// TIA Portal V16 export
// export: Created 2022-07-21T09:35:35.040371Z, ExportSetting WithDefaults, DisplayName Totally Integrated Automation Portal, DisplayVersion V16 Update 4, DisplayName TIA Portal Version Control Interface, DisplayVersion V16 Update 2, DisplayName TIA Portal Openness, DisplayVersion V16 Update 4, DisplayName SINAMICS Startdrive Advanced, DisplayVersion V16 Update 5, DisplayName SINAMICS Startdrive G130, G150, S120, S150, SINAMICS MV, S210, DisplayVersion V16 Update 5, DisplayName SINAMICS Startdrive G110M, G120, G120C, G120D, G120P, G115D, DisplayVersion V16 Update 5, DisplayName STEP 7 Professional, DisplayVersion V16 Update 4, DisplayName STEP 7 Safety, DisplayVersion V16, DisplayName WinCC Advanced, DisplayVersion V16 Update 4
FUNCTION_BLOCK "fbValve"   // FB702, LAD
TITLE = Valve / Obsługa zaworu
{ S7_Optimized_Access := 'TRUE' }
AUTHOR : a32thzz
VERSION : 0.1
// In this block alarms, statuses and commands for electrovalves are generated / Ten blok służy do generowania alarmów, statusów i wysyłania komend dla siłowników kontrolowanych przez elektrozawory.
// stored: AutoNumber false, IsIECCheckEnabled false, IsRetainMemResEnabled false, MemoryReserve 100, SetENOAutomatically false, UDAEnableTagReadback false
   VAR_INPUT
      inPeripheryOK : Bool;   // Zezwolenie od peryferiów (PN, Elektryka)
      inHomeLS : Bool;   // Czujnik pozycji bazowej / Home position sensor
      inWorkLS : Bool;   // Czujnik pozycji roboczej / Work position sensor
      inAutoHome : Bool;   // Krok sekwencji "do pozycji bazowej" / Move to home position
      inAutoWork : Bool;   // Krok sekwencji "do pozycji roboczej" / Move to work position
      inHold : Bool := true;   // Podtrzymanie zasilania elektrozaworu podczas ruchu do pozycji / Hold electrovalve power supply during movement
      inJog : Bool := true;   // Podtrzymanie zasilania elektrozaworu po osiągnięciu pozycji końcowej / Hold electrovalve power supply after reaching position
      inDelayPTAlm0 : Time := T#1s;   // Czas opóźnienia dla alarmu 0 / alarm delay 0
      inDelayPTAlm1 : Time := T#1s;   // Czas opóźnienia dla alarmu 1 / alarm delay 1
      inDelayPTAlm2 : Time := T#1s;   // Czas opóźnienia dla alarmu 2 / alarm delay 2
      inDelayPTAlm3 : Time := T#1s;   // Czas opóźnienia dla alarmu 3 / alarm delay 3
      inDelayPTAlm4 : Time := T#1s;   // Czas opóźnienia dla alarmu 4 / alarm delay 4
      inDelayPTAlm5 : Time := T#1s;   // Czas opóźnienia dla alarmu 5 / alarm delay 5
      inAlmMask : Word := W#16#FFE0;   // Maskowanie alarmów
      inGroup : "typeGroup";   // Grupa do której przypisany jest zawór / Valve group
   END_VAR
   VAR_OUTPUT
      ouHomeSV : Bool;   // Elektrozawór dla pozycji bazowej / Electrovalve to home porisiton
      ouWorkSV : Bool;   // Elektrozawór dla pozycji roboczej / Electrovalve to work porisiton
   END_VAR
   VAR_IN_OUT
      ioValve : "typeValve";
   END_VAR
   VAR
      instTmrDlyHome { S7_SetPoint := 'True'} : TON_TIME;   // Opóźnienie dla symulacji ruchu do pozycji bazowej / Delay move to home position
      instTmrDlyWork { S7_SetPoint := 'True'} : TON_TIME;   // Opóźnienie dla symulacji ruchu do pozycji roboczej / Delay move to work position
      instReset { S7_SetPoint := 'True'} : "fbReset";
      instAlm { S7_SetPoint := 'True'} : Array[0..15] of "fbAlarmMessage";
   END_VAR
   // instTmrDlyHome.PT := T#0ms;
   // instTmrDlyWork.PT := T#0ms;
BEGIN

REGION Network 1: Home position sensor / Czujnik pozycji bazowej
   // If home position sensor is not active, input is simulated after output activation and delay time / Jeśli czujnik pozycji bazowej został wyłączony wejście jest symulowane po aktywacji wyjścia i upłynięciu zdefiniowanego czasu.
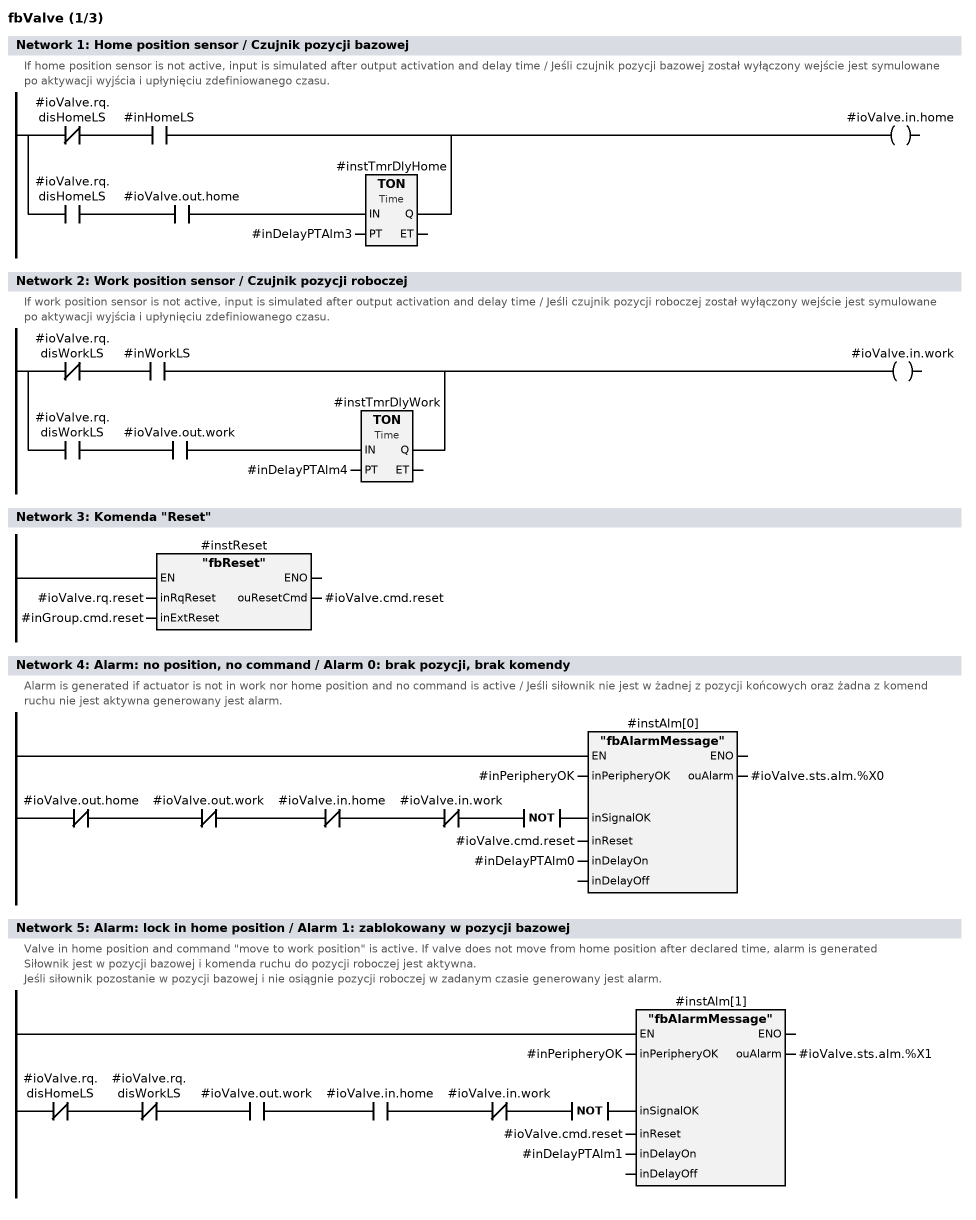
   RUNG wire#powerrail
      I_Contact( #ioValve.rq.disHomeLS )
      Contact( #inHomeLS )
      wire#w1
      Coil( #ioValve.in.home )
   END_RUNG
   RUNG wire#powerrail
      Contact( #ioValve.rq.disHomeLS )
      Contact( #ioValve.out.home )
      { S7_Templates := "time_type := Time" } #instTmrDlyHome.TON(pt := #inDelayPTAlm3, et =>)
   END_RUNG wire#w1
   // the same network as SCL:
   #instTmrDlyHome(IN := #ioValve.rq.disHomeLS AND #ioValve.out.home, PT := #inDelayPTAlm3);   // TON
   #ioValve.in.home := (NOT #ioValve.rq.disHomeLS AND #inHomeLS) OR #instTmrDlyHome.Q;
END_REGION

REGION Network 2: Work position sensor / Czujnik pozycji roboczej
   // If work position sensor is not active, input is simulated after output activation and delay time / Jeśli czujnik pozycji roboczej został wyłączony wejście jest symulowane po aktywacji wyjścia i upłynięciu zdefiniowanego czasu.
   RUNG wire#powerrail
      I_Contact( #ioValve.rq.disWorkLS )
      Contact( #inWorkLS )
      wire#w1
      Coil( #ioValve.in.work )
   END_RUNG
   RUNG wire#powerrail
      Contact( #ioValve.rq.disWorkLS )
      Contact( #ioValve.out.work )
      { S7_Templates := "time_type := Time" } #instTmrDlyWork.TON(pt := #inDelayPTAlm4, et =>)
   END_RUNG wire#w1
   // the same network as SCL:
   #instTmrDlyWork(IN := #ioValve.rq.disWorkLS AND #ioValve.out.work, PT := #inDelayPTAlm4);   // TON
   #ioValve.in.work := (NOT #ioValve.rq.disWorkLS AND #inWorkLS) OR #instTmrDlyWork.Q;
END_REGION

REGION Network 3: Komenda "Reset"
   RUNG wire#powerrail
      #instReset(inRqReset := #ioValve.rq.reset, inExtReset := #inGroup.cmd.reset, ouResetCmd => #ioValve.cmd.reset)
   END_RUNG
   // the same network as SCL:
   #instReset(inRqReset := #ioValve.rq.reset,   // "fbReset"
              inExtReset := #inGroup.cmd.reset,
              ouResetCmd => #ioValve.cmd.reset);
END_REGION

REGION Network 4: Alarm: no position, no command / Alarm 0: brak pozycji, brak komendy
   // Alarm is generated if actuator is not in work nor home position and no command is active / Jeśli siłownik nie jest w żadnej z pozycji końcowych oraz żadna z komend ruchu nie jest aktywna generowany jest alarm.
   RUNG wire#powerrail
      #instAlm[0](inSignalOK := wire#w1, inPeripheryOK := #inPeripheryOK, inReset := #ioValve.cmd.reset, inDelayOn := #inDelayPTAlm0, inDelayOff :=, ouAlarm => #ioValve.sts.alm.%X0)
   END_RUNG
   RUNG wire#powerrail
      I_Contact( #ioValve.out.home )
      I_Contact( #ioValve.out.work )
      I_Contact( #ioValve.in.home )
      I_Contact( #ioValve.in.work )
      Not()
   END_RUNG wire#w1
   // the same network as SCL:
   #instAlm[0](inPeripheryOK := #inPeripheryOK,   // "fbAlarmMessage"
               inSignalOK := NOT (NOT #ioValve.out.home AND NOT #ioValve.out.work AND NOT #ioValve.in.home AND NOT #ioValve.in.work),
               inReset := #ioValve.cmd.reset,
               inDelayOn := #inDelayPTAlm0,
               ouAlarm => #ioValve.sts.alm.%X0);
END_REGION

REGION Network 5: Alarm: lock in home position / Alarm 1: zablokowany w pozycji bazowej
   // Valve in home position and command "move to work position" is active. If valve does not move from home position after declared time, alarm is generated
   // Siłownik jest w pozycji bazowej i komenda ruchu do pozycji roboczej jest aktywna.
   // Jeśli siłownik pozostanie w pozycji bazowej i nie osiągnie pozycji roboczej w zadanym czasie generowany jest alarm.
   RUNG wire#powerrail
      #instAlm[1](inSignalOK := wire#w1, inPeripheryOK := #inPeripheryOK, inReset := #ioValve.cmd.reset, inDelayOn := #inDelayPTAlm1, inDelayOff :=, ouAlarm => #ioValve.sts.alm.%X1)
   END_RUNG
   RUNG wire#powerrail
      I_Contact( #ioValve.rq.disHomeLS )
      I_Contact( #ioValve.rq.disWorkLS )
      Contact( #ioValve.out.work )
      Contact( #ioValve.in.home )
      I_Contact( #ioValve.in.work )
      Not()
   END_RUNG wire#w1
   // the same network as SCL:
   #instAlm[1](inPeripheryOK := #inPeripheryOK,   // "fbAlarmMessage"
               inSignalOK := NOT (NOT #ioValve.rq.disHomeLS AND NOT #ioValve.rq.disWorkLS AND #ioValve.out.work AND #ioValve.in.home AND NOT #ioValve.in.work),
               inReset := #ioValve.cmd.reset,
               inDelayOn := #inDelayPTAlm1,
               ouAlarm => #ioValve.sts.alm.%X1);
END_REGION

REGION Network 6: Alarm: lock in work position / Alarm 2: zablokowany w pozycji roboczej
   // Valve in work position and command "move to home position" is active. If valve does not move from work position after declared time, alarm is generated
   // Siłownik jest w pozycji roboczej i komenda ruchu do pozycji bazowej jest aktywna.
   // Jeśli siłownik pozostanie w pozycji roboczej i nie osiągnie pozycji bazowej w zadanym czasie generowany jest alarm.
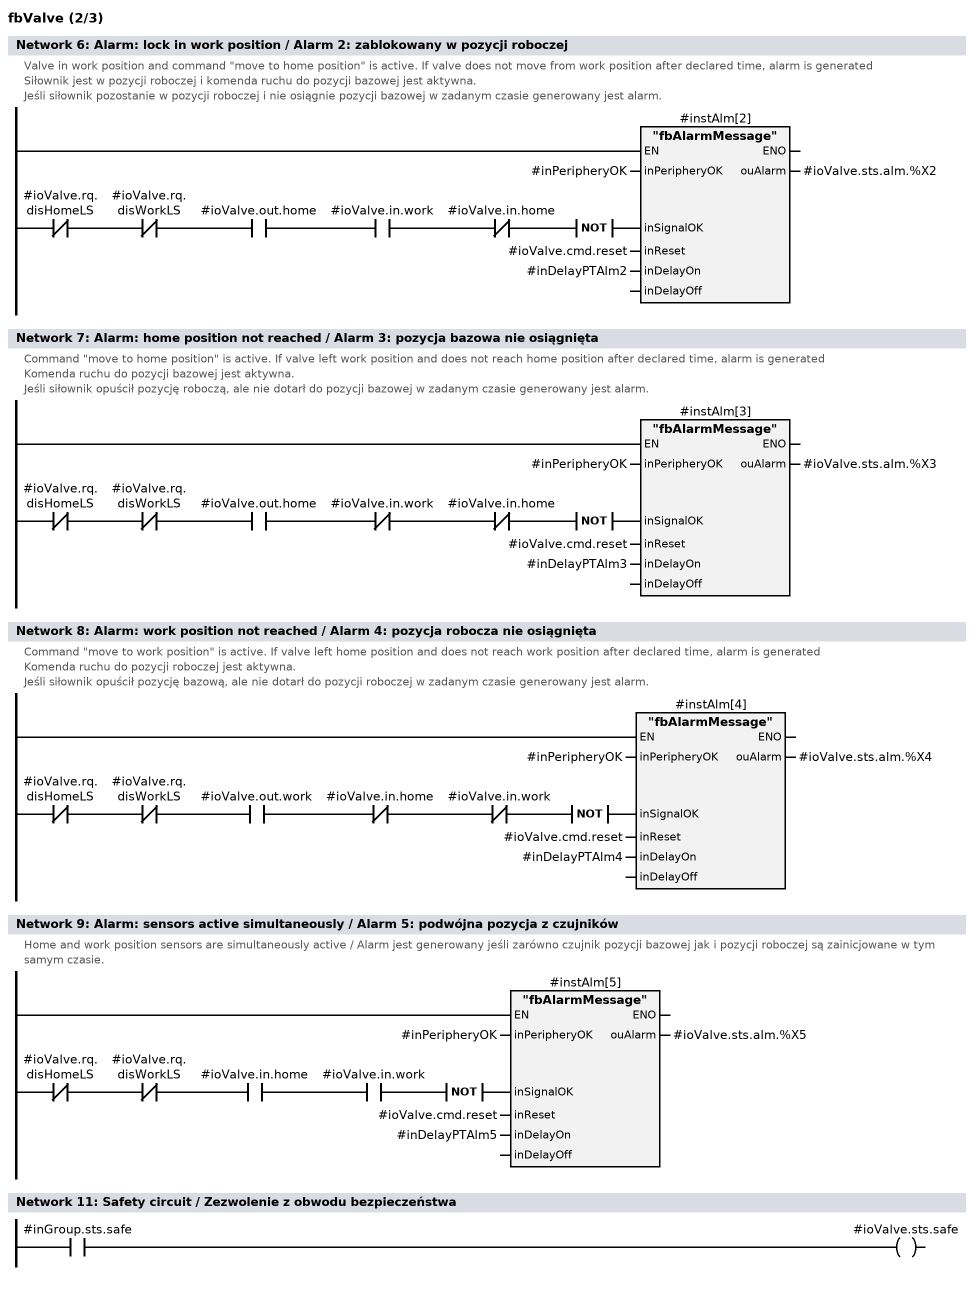
   RUNG wire#powerrail
      #instAlm[2](inSignalOK := wire#w1, inPeripheryOK := #inPeripheryOK, inReset := #ioValve.cmd.reset, inDelayOn := #inDelayPTAlm2, inDelayOff :=, ouAlarm => #ioValve.sts.alm.%X2)
   END_RUNG
   RUNG wire#powerrail
      I_Contact( #ioValve.rq.disHomeLS )
      I_Contact( #ioValve.rq.disWorkLS )
      Contact( #ioValve.out.home )
      Contact( #ioValve.in.work )
      I_Contact( #ioValve.in.home )
      Not()
   END_RUNG wire#w1
   // the same network as SCL:
   #instAlm[2](inPeripheryOK := #inPeripheryOK,   // "fbAlarmMessage"
               inSignalOK := NOT (NOT #ioValve.rq.disHomeLS AND NOT #ioValve.rq.disWorkLS AND #ioValve.out.home AND #ioValve.in.work AND NOT #ioValve.in.home),
               inReset := #ioValve.cmd.reset,
               inDelayOn := #inDelayPTAlm2,
               ouAlarm => #ioValve.sts.alm.%X2);
END_REGION

REGION Network 7: Alarm: home position not reached / Alarm 3: pozycja bazowa nie osiągnięta
   // Command "move to home position" is active. If valve left work position and does not reach home position after declared time, alarm is generated
   // Komenda ruchu do pozycji bazowej jest aktywna.
   // Jeśli siłownik opuścił pozycję roboczą, ale nie dotarł do pozycji bazowej w zadanym czasie generowany jest alarm.
   RUNG wire#powerrail
      #instAlm[3](inSignalOK := wire#w1, inPeripheryOK := #inPeripheryOK, inReset := #ioValve.cmd.reset, inDelayOn := #inDelayPTAlm3, inDelayOff :=, ouAlarm => #ioValve.sts.alm.%X3)
   END_RUNG
   RUNG wire#powerrail
      I_Contact( #ioValve.rq.disHomeLS )
      I_Contact( #ioValve.rq.disWorkLS )
      Contact( #ioValve.out.home )
      I_Contact( #ioValve.in.work )
      I_Contact( #ioValve.in.home )
      Not()
   END_RUNG wire#w1
   // the same network as SCL:
   #instAlm[3](inPeripheryOK := #inPeripheryOK,   // "fbAlarmMessage"
               inSignalOK := NOT (NOT #ioValve.rq.disHomeLS AND NOT #ioValve.rq.disWorkLS AND #ioValve.out.home AND NOT #ioValve.in.work AND NOT #ioValve.in.home),
               inReset := #ioValve.cmd.reset,
               inDelayOn := #inDelayPTAlm3,
               ouAlarm => #ioValve.sts.alm.%X3);
END_REGION

REGION Network 8: Alarm: work position not reached / Alarm 4: pozycja robocza nie osiągnięta
   // Command "move to work position" is active. If valve left home position and does not reach work position after declared time, alarm is generated
   // Komenda ruchu do pozycji roboczej jest aktywna.
   // Jeśli siłownik opuścił pozycję bazową, ale nie dotarł do pozycji roboczej w zadanym czasie generowany jest alarm.
   RUNG wire#powerrail
      #instAlm[4](inSignalOK := wire#w1, inPeripheryOK := #inPeripheryOK, inReset := #ioValve.cmd.reset, inDelayOn := #inDelayPTAlm4, inDelayOff :=, ouAlarm => #ioValve.sts.alm.%X4)
   END_RUNG
   RUNG wire#powerrail
      I_Contact( #ioValve.rq.disHomeLS )
      I_Contact( #ioValve.rq.disWorkLS )
      Contact( #ioValve.out.work )
      I_Contact( #ioValve.in.home )
      I_Contact( #ioValve.in.work )
      Not()
   END_RUNG wire#w1
   // the same network as SCL:
   #instAlm[4](inPeripheryOK := #inPeripheryOK,   // "fbAlarmMessage"
               inSignalOK := NOT (NOT #ioValve.rq.disHomeLS AND NOT #ioValve.rq.disWorkLS AND #ioValve.out.work AND NOT #ioValve.in.home AND NOT #ioValve.in.work),
               inReset := #ioValve.cmd.reset,
               inDelayOn := #inDelayPTAlm4,
               ouAlarm => #ioValve.sts.alm.%X4);
END_REGION

REGION Network 9: Alarm: sensors active simultaneously / Alarm 5: podwójna pozycja z czujników
   // Home and work position sensors are simultaneously active / Alarm jest generowany jeśli zarówno czujnik pozycji bazowej jak i pozycji roboczej są zainicjowane w tym samym czasie.
   RUNG wire#powerrail
      #instAlm[5](inSignalOK := wire#w1, inPeripheryOK := #inPeripheryOK, inReset := #ioValve.cmd.reset, inDelayOn := #inDelayPTAlm5, inDelayOff :=, ouAlarm => #ioValve.sts.alm.%X5)
   END_RUNG
   RUNG wire#powerrail
      I_Contact( #ioValve.rq.disHomeLS )
      I_Contact( #ioValve.rq.disWorkLS )
      Contact( #ioValve.in.home )
      Contact( #ioValve.in.work )
      Not()
   END_RUNG wire#w1
   // the same network as SCL:
   #instAlm[5](inPeripheryOK := #inPeripheryOK,   // "fbAlarmMessage"
               inSignalOK := NOT (NOT #ioValve.rq.disHomeLS AND NOT #ioValve.rq.disWorkLS AND #ioValve.in.home AND #ioValve.in.work),
               inReset := #ioValve.cmd.reset,
               inDelayOn := #inDelayPTAlm5,
               ouAlarm => #ioValve.sts.alm.%X5);
END_REGION

REGION Network 10 (SCL): Status: noAlm
   #ioValve.sts.noAlm := (#ioValve.sts.alm AND NOT #inAlmMask) = 0;
END_REGION

REGION Network 11: Safety circuit / Zezwolenie z obwodu bezpieczeństwa
   RUNG wire#powerrail
      Contact( #inGroup.sts.safe )
      Coil( #ioValve.sts.safe )
   END_RUNG
   // the same network as SCL:
   #ioValve.sts.safe := #inGroup.sts.safe;
END_REGION

REGION Network 12: Necessary conditions met / Warunki konieczne spełnione
   // Necessary conditions / Warunki konieczne: obwód bezpieczeństwa musi byś zresetowany i nie ma aktywnych alarmów
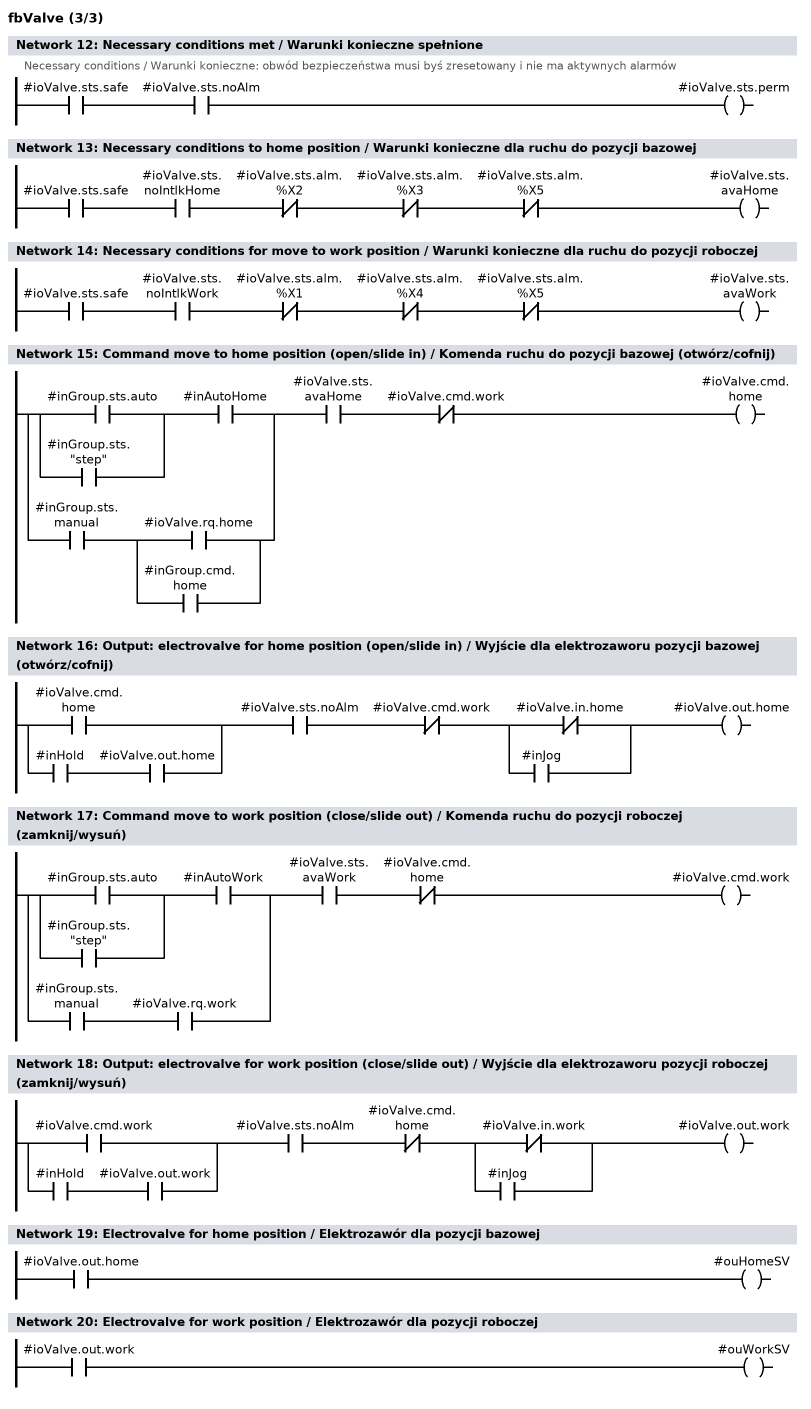
   RUNG wire#powerrail
      Contact( #ioValve.sts.safe )
      Contact( #ioValve.sts.noAlm )
      Coil( #ioValve.sts.perm )
   END_RUNG
   // the same network as SCL:
   #ioValve.sts.perm := #ioValve.sts.safe AND #ioValve.sts.noAlm;
END_REGION

REGION Network 13: Necessary conditions to home position / Warunki konieczne dla ruchu do pozycji bazowej
   RUNG wire#powerrail
      Contact( #ioValve.sts.safe )
      Contact( #ioValve.sts.noIntlkHome )
      I_Contact( #ioValve.sts.alm.%X2 )
      I_Contact( #ioValve.sts.alm.%X3 )
      I_Contact( #ioValve.sts.alm.%X5 )
      Coil( #ioValve.sts.avaHome )
   END_RUNG
   // the same network as SCL:
   #ioValve.sts.avaHome := #ioValve.sts.safe AND #ioValve.sts.noIntlkHome AND NOT #ioValve.sts.alm.%X2 AND NOT #ioValve.sts.alm.%X3 AND NOT #ioValve.sts.alm.%X5;
END_REGION

REGION Network 14: Necessary conditions for move to work position / Warunki konieczne dla ruchu do pozycji roboczej
   RUNG wire#powerrail
      Contact( #ioValve.sts.safe )
      Contact( #ioValve.sts.noIntlkWork )
      I_Contact( #ioValve.sts.alm.%X1 )
      I_Contact( #ioValve.sts.alm.%X4 )
      I_Contact( #ioValve.sts.alm.%X5 )
      Coil( #ioValve.sts.avaWork )
   END_RUNG
   // the same network as SCL:
   #ioValve.sts.avaWork := #ioValve.sts.safe AND #ioValve.sts.noIntlkWork AND NOT #ioValve.sts.alm.%X1 AND NOT #ioValve.sts.alm.%X4 AND NOT #ioValve.sts.alm.%X5;
END_REGION

REGION Network 15: Command move to home position (open/slide in) / Komenda ruchu do pozycji bazowej (otwórz/cofnij)
   RUNG wire#powerrail
      Contact( #inGroup.sts.auto )
      wire#w1
      Contact( #inAutoHome )
      wire#w2
      Contact( #ioValve.sts.avaHome )
      I_Contact( #ioValve.cmd.work )
      Coil( #ioValve.cmd.home )
   END_RUNG
   RUNG wire#powerrail
      Contact( #inGroup.sts."step" )
   END_RUNG wire#w1
   RUNG wire#powerrail
      Contact( #inGroup.sts.manual )
      wire#w3
      Contact( #ioValve.rq.home )
   END_RUNG wire#w2
   RUNG wire#w3
      Contact( #inGroup.cmd.home )
   END_RUNG wire#w2
   // the same network as SCL:
   #ioValve.cmd.home := (((#inGroup.sts.auto OR #inGroup.sts."step") AND #inAutoHome) OR (#inGroup.sts.manual AND (#ioValve.rq.home OR #inGroup.cmd.home))) AND #ioValve.sts.avaHome AND NOT #ioValve.cmd.work;
END_REGION

REGION Network 16: Output: electrovalve for home position (open/slide in) / Wyjście dla elektrozaworu pozycji bazowej (otwórz/cofnij)
   RUNG wire#powerrail
      Contact( #ioValve.cmd.home )
      wire#w1
      Contact( #ioValve.sts.noAlm )
      I_Contact( #ioValve.cmd.work )
      wire#w2
      I_Contact( #ioValve.in.home )
      wire#w3
      Coil( #ioValve.out.home )
   END_RUNG
   RUNG wire#powerrail
      Contact( #inHold )
      Contact( #ioValve.out.home )
   END_RUNG wire#w1
   RUNG wire#w2
      Contact( #inJog )
   END_RUNG wire#w3
   // the same network as SCL:
   #ioValve.out.home := (#ioValve.cmd.home OR (#inHold AND #ioValve.out.home)) AND #ioValve.sts.noAlm AND NOT #ioValve.cmd.work AND (NOT #ioValve.in.home OR #inJog);
END_REGION

REGION Network 17: Command move to work position (close/slide out) / Komenda ruchu do pozycji roboczej (zamknij/wysuń)
   RUNG wire#powerrail
      Contact( #inGroup.sts.auto )
      wire#w1
      Contact( #inAutoWork )
      wire#w2
      Contact( #ioValve.sts.avaWork )
      I_Contact( #ioValve.cmd.home )
      Coil( #ioValve.cmd.work )
   END_RUNG
   RUNG wire#powerrail
      Contact( #inGroup.sts."step" )
   END_RUNG wire#w1
   RUNG wire#powerrail
      Contact( #inGroup.sts.manual )
      Contact( #ioValve.rq.work )
   END_RUNG wire#w2
   // the same network as SCL:
   #ioValve.cmd.work := (((#inGroup.sts.auto OR #inGroup.sts."step") AND #inAutoWork) OR (#inGroup.sts.manual AND #ioValve.rq.work)) AND #ioValve.sts.avaWork AND NOT #ioValve.cmd.home;
END_REGION

REGION Network 18: Output: electrovalve for work position (close/slide out) / Wyjście dla elektrozaworu pozycji roboczej (zamknij/wysuń)
   RUNG wire#powerrail
      Contact( #ioValve.cmd.work )
      wire#w1
      Contact( #ioValve.sts.noAlm )
      I_Contact( #ioValve.cmd.home )
      wire#w2
      I_Contact( #ioValve.in.work )
      wire#w3
      Coil( #ioValve.out.work )
   END_RUNG
   RUNG wire#powerrail
      Contact( #inHold )
      Contact( #ioValve.out.work )
   END_RUNG wire#w1
   RUNG wire#w2
      Contact( #inJog )
   END_RUNG wire#w3
   // the same network as SCL:
   #ioValve.out.work := (#ioValve.cmd.work OR (#inHold AND #ioValve.out.work)) AND #ioValve.sts.noAlm AND NOT #ioValve.cmd.home AND (NOT #ioValve.in.work OR #inJog);
END_REGION

REGION Network 19: Electrovalve for home position / Elektrozawór dla pozycji bazowej
   RUNG wire#powerrail
      Contact( #ioValve.out.home )
      Coil( #ouHomeSV )
   END_RUNG
   // the same network as SCL:
   #ouHomeSV := #ioValve.out.home;
END_REGION

REGION Network 20: Electrovalve for work position / Elektrozawór dla pozycji roboczej
   RUNG wire#powerrail
      Contact( #ioValve.out.work )
      Coil( #ouWorkSV )
   END_RUNG
   // the same network as SCL:
   #ouWorkSV := #ioValve.out.work;
END_REGION
END_FUNCTION_BLOCK
